(* IEC 61131-3 sources: plc-st-review/examples/state-machine, 14 files *)

(* ---- E_ConveyorState.st ---- *)
(*
 * Conveyor state machine enum.
 *
 * Used by FB_ConveyorState and (separately) by Conveyor_HMI. If we add a
 * value here and forget to handle it in the HMI's CASE, plc-st-review will
 * surface STATE_UNHANDLED.
 *)

TYPE E_ConveyorState :
    (IDLE := 0, STARTING, RUNNING, STOPPING, FAULT);
END_TYPE

(* ---- E_DiagMode.st ---- *)
(*
 * E_DiagMode — diagnostic verbosity levels for FB_AxisRamp.
 *
 * The demo PR removes DIAG_LEGACY (ENUM_VALUE_REMOVED) and drops the
 * DIAG_VERBOSE branch from FB_AxisRamp's CASE while keeping the value
 * in the enum (ENUM_VALUE_UNUSED).
 *)

TYPE E_DiagMode :
    (DIAG_OFF := 0, DIAG_BASIC, DIAG_VERBOSE, DIAG_LEGACY);
END_TYPE

(* ---- Globals.st ---- *)
(*
 * Globals for the conveyor demo.
 *
 * Demonstrates VAR_GLOBAL CONSTANT (constants the engine watches) and a
 * non-constant global (typed reference for callers).
 *)

VAR_GLOBAL CONSTANT
    SAFETY_TIMEOUT      : TIME := T#2s;
    LIMIT_MAX_SPEED     : INT  := 100;
    LIMIT_MIN_SPEED     : INT  := 5;
    CONVEYOR_SLOTS      : INT  := 10;
END_VAR

VAR_GLOBAL
    gFlowSetpoint       : REAL := 0.0;
END_VAR

(* ---- I_Diagnostic.st ---- *)
(*
 * I_Diagnostic — diagnostic contract implemented by FB_DiagUnit.
 *
 * The demo PR adds a second method (SelfTest) to this interface without
 * adding it to the implementer, surfacing METHOD_ADDED_TO_INTERFACE.
 *)

INTERFACE I_Diagnostic
METHOD Reset : BOOL
END_METHOD
END_INTERFACE

(* ---- FB_AxisRamp.st ---- *)
{attribute 'qualified_only'}
(*
 * FB_AxisRamp — ramps an axis toward a setpoint and counts cycles.
 *
 * The demo PR exercises five diff-based checks against this file:
 *   PRAGMA_CHANGED         the {attribute} pragma is swapped
 *   INHERITANCE_CHANGED    EXTENDS FB_Base -> FB_BaseV2
 *   ARRAY_BOUNDS_CHANGED   aHistory grows from [0..9] to [0..19]
 *   COUNTER_VALUE_CHANGED  cCycles.PV 100 -> 500
 *   ENUM_VALUE_UNUSED      the DIAG_VERBOSE CASE branch is removed
 *)

FUNCTION_BLOCK FB_AxisRamp EXTENDS FB_Base
VAR_INPUT
    rSetpoint : REAL;
    eMode     : E_DiagMode;
    xCount    : BOOL;
END_VAR
VAR_OUTPUT
    rPosition : REAL;
END_VAR
VAR
    aHistory  : ARRAY [0..9] OF REAL;
    cCycles   : CTU;
    iIndex    : INT;
END_VAR

cCycles(CU := xCount, PV := 100);

CASE eMode OF
    E_DiagMode.DIAG_OFF:
        rPosition := rSetpoint;
    E_DiagMode.DIAG_BASIC:
        rPosition := rSetpoint * 0.5;
    E_DiagMode.DIAG_VERBOSE:
        rPosition := rSetpoint * 0.25;
    E_DiagMode.DIAG_LEGACY:
        rPosition := 0.0;
END_CASE;

aHistory[iIndex] := rSetpoint;
END_FUNCTION_BLOCK

(* ---- FB_Base.st ---- *)
(*
 * FB_Base / FB_BaseV2 — base classes for the diagnostics demo.
 *
 * FB_AxisRamp EXTENDS FB_Base here; the demo PR re-points it at
 * FB_BaseV2 to surface INHERITANCE_CHANGED. Both are deliberately
 * trivial — they exist only to be inherited from.
 *)

FUNCTION_BLOCK FB_Base
VAR
    xInitialized : BOOL;
END_VAR
xInitialized := TRUE;
END_FUNCTION_BLOCK

FUNCTION_BLOCK FB_BaseV2
VAR
    xInitialized : BOOL;
    iRevision    : INT;
END_VAR
xInitialized := TRUE;
iRevision := 2;
END_FUNCTION_BLOCK

(* ---- FB_ConveyorState.st ---- *)
(*
 * FB_ConveyorState — minimal conveyor state machine.
 *
 * Implements a Mealy-style state machine over E_ConveyorState, with a
 * startup-delay timer and a configurable target speed. Designed to exercise
 * several plc-st-review checks at once when the file is edited.
 *)

FUNCTION_BLOCK FB_ConveyorState
VAR_INPUT
    xEnable             : BOOL;
    rTargetSpeed        : REAL;
END_VAR
VAR_OUTPUT
    eState              : E_ConveyorState;
    xRunning            : BOOL;
    rActualSpeed        : REAL;
END_VAR
VAR
    T_StartupDelay      : TON;
    iRamp               : INT;
END_VAR

(* Startup delay — driven by a TON instance. *)
T_StartupDelay(IN := (eState = E_ConveyorState.STARTING), PT := T#2s);

CASE eState OF
    E_ConveyorState.IDLE:
        IF xEnable THEN
            eState := E_ConveyorState.STARTING;
        END_IF;

    E_ConveyorState.STARTING:
        IF T_StartupDelay.Q THEN
            eState := E_ConveyorState.RUNNING;
            rActualSpeed := 0.0;
        END_IF;

    E_ConveyorState.RUNNING:
        xRunning := TRUE;
        (* Linear ramp toward target speed using a FOR loop. *)
        FOR iRamp := 1 TO CONVEYOR_SLOTS BY 1 DO
            rActualSpeed := rActualSpeed + (rTargetSpeed - rActualSpeed) * 0.1;
        END_FOR;
        IF NOT xEnable THEN
            eState := E_ConveyorState.STOPPING;
        END_IF;

    E_ConveyorState.STOPPING:
        xRunning := FALSE;
        rActualSpeed := 0.0;
        eState := E_ConveyorState.IDLE;

    E_ConveyorState.FAULT:
        xRunning := FALSE;
        rActualSpeed := 0.0;
END_CASE;

END_FUNCTION_BLOCK

(* ---- FB_DiagUnit.st ---- *)
(*
 * FB_DiagUnit — implements I_Diagnostic.
 *
 * The demo PR adds a SelfTest method to I_Diagnostic; this FB does NOT
 * gain a matching method, surfacing METHOD_ADDED_TO_INTERFACE.
 *)

FUNCTION_BLOCK FB_DiagUnit IMPLEMENTS I_Diagnostic
VAR
    xReady : BOOL;
END_VAR

METHOD Reset : BOOL
    xReady := FALSE;
    Reset := TRUE;
END_METHOD

xReady := TRUE;
END_FUNCTION_BLOCK

(* ---- FB_Legacy.st ---- *)
(*
 * FB_Legacy — a deprecated helper kept only so the demo PR can delete
 * the whole file and surface POU_DELETED. Nothing calls it.
 *)

FUNCTION_BLOCK FB_Legacy
VAR_INPUT
    xTrigger : BOOL;
END_VAR
VAR_OUTPUT
    xDone : BOOL;
END_VAR
xDone := xTrigger;
END_FUNCTION_BLOCK

(* ---- FB_LineController.st ---- *)
(*
 * FB_LineController - top-level conveyor-line coordinator.
 *
 * A deliberately involved orchestrator: it sequences the axis ramp, the speed
 * estimate, the diagnostic unit and the metrics helper behind layered mode and
 * guard logic. It exists so the --metrics report has a realistic
 * high-complexity hub to rank (it lands in the red band), and so the blocks it
 * drives are reported as live rather than dead code. The body is intentionally
 * tangled but otherwise clean - it triggers no review findings on its own.
 *)

FUNCTION_BLOCK FB_LineController EXTENDS FB_BaseV2
VAR_INPUT
    xRun        : BOOL;
    iMode       : INT;
    rSetpoint   : REAL;
    iPulses     : INT;
    xManual     : BOOL;
END_VAR
VAR_OUTPUT
    rLineSpeed  : REAL;
    xActive     : BOOL;
    iFaultCode  : INT;
END_VAR
VAR
    fbRamp      : FB_AxisRamp;
    fbSpeed     : FB_SpeedCalc;
    fbDiag      : FB_DiagUnit;
    fbMetrics   : FB_MetricsDemo;
    T_Settle    : TON;
    rLocalSpeed : REAL;
    iStep       : INT;
    iGuard      : INT;
    iFault      : INT;
END_VAR

(* Sub-blocks run every scan; their outputs feed the mode logic below. *)
fbSpeed(iPulseCount := iPulses, rScale := 0.5);
fbDiag();
T_Settle(IN := xRun, PT := T#500ms);

CASE iMode OF
    0:  (* idle - wait for a run request that isn't a manual hold *)
        IF xRun AND NOT xManual THEN
            iStep := 1;
        ELSIF xManual THEN
            iStep := 0;
        END_IF;

    1:  (* ramping - climb toward setpoint once the settle timer elapses *)
        IF T_Settle.Q THEN
            fbRamp(rSetpoint := rSetpoint, eMode := E_DiagMode.DIAG_BASIC, xCount := xRun);
            FOR iGuard := 1 TO CONVEYOR_SLOTS BY 1 DO
                IF fbSpeed.rSpeed > rLocalSpeed THEN
                    rLocalSpeed := rLocalSpeed + (rSetpoint - rLocalSpeed) * 0.1;
                    IF rLocalSpeed > LIMIT_MAX_SPEED THEN
                        rLocalSpeed := LIMIT_MAX_SPEED;
                    END_IF;
                    IF xManual OR iGuard > LIMIT_MIN_SPEED THEN
                        iStep := iGuard;
                    END_IF;
                END_IF;
            END_FOR;
        END_IF;

    2:  (* running - advance the line, sampling metrics as it goes *)
        WHILE iStep < CONVEYOR_SLOTS AND xRun DO
            iStep := iStep + 1;
            IF rLocalSpeed >= rSetpoint THEN
                EXIT;
            END_IF;
            IF iStep >= LIMIT_MIN_SPEED THEN
                fbMetrics(x := iStep);
                IF fbMetrics.y > 0 OR xManual THEN
                    rLocalSpeed := fbRamp.rPosition;
                END_IF;
            END_IF;
        END_WHILE;

    3:  (* diagnostics - classify the speed estimate into a fault code *)
        IF fbSpeed.rSpeed < LIMIT_MIN_SPEED THEN
            iFault := 1;
        ELSIF fbSpeed.rSpeed > LIMIT_MAX_SPEED THEN
            iFault := 2;
        ELSE
            iFault := 0;
        END_IF;

    4:  (* hold - manual override parks the line *)
        IF xManual THEN
            iStep := 0;
            rLocalSpeed := 0.0;
        END_IF;

    ELSE
        iStep := 0;
END_CASE;

IF iFault > 0 THEN
    xActive := FALSE;
ELSIF xRun THEN
    xActive := TRUE;
END_IF;

rLineSpeed := rLocalSpeed;
iFaultCode := iFault;
END_FUNCTION_BLOCK

(* ---- FB_MetricsDemo.st ---- *)
// Baseline version of the metrics-demo block. The demo PR (#1) ships a
// heavily expanded version of this same FB, so the diff exercises the
// metric-regression checks (COMPLEXITY_INCREASED, NESTING_INCREASED,
// LOC_SPIKE) without disturbing any other fixture.
FUNCTION_BLOCK FB_MetricsDemo
VAR_INPUT
    x : INT;
END_VAR
VAR_OUTPUT
    y : INT;
END_VAR
y := x;
END_FUNCTION_BLOCK

(* ---- FB_SpeedCalc.st ---- *)
(*
 * FB_SpeedCalc — converts a raw pulse count to a speed estimate.
 *
 * The demo PR renames this POU to FB_SpeedCalculator (keeping the exact
 * same input/output signature) to surface POU_RENAMED.
 *)

FUNCTION_BLOCK FB_SpeedCalc
VAR_INPUT
    iPulseCount : INT;
    rScale      : REAL;
END_VAR
VAR_OUTPUT
    rSpeed      : REAL;
END_VAR
VAR
    rRaw        : REAL;
END_VAR
rRaw := rScale;
IF iPulseCount > 0 THEN
    rSpeed := rRaw;
ELSE
    rSpeed := 0.0;
END_IF;
END_FUNCTION_BLOCK

(* ---- FB_Watchdog.st ---- *)
(*
 * FB_Watchdog — trivial heartbeat monitor.
 *
 * The demo PR changes ONLY the inline comment below, leaving the AST
 * structurally identical between revisions, to surface COMMENT_ONLY.
 *)

FUNCTION_BLOCK FB_Watchdog
VAR_INPUT
    xHeartbeat : BOOL;
END_VAR
VAR_OUTPUT
    xAlive : BOOL;
END_VAR
(* heartbeat is forwarded straight through *)
xAlive := xHeartbeat;
END_FUNCTION_BLOCK

(* ---- Conveyor_HMI.st ---- *)
(*
 * Conveyor_HMI — display formatter for the conveyor state machine.
 *
 * Lives in a different file than FB_ConveyorState on purpose: the engine's
 * cross-file analysis is what surfaces STATE_UNHANDLED when the enum gains
 * a value and only one of the CASE statements is updated.
 *)

PROGRAM Conveyor_HMI
VAR
    fbConveyor          : FB_ConveyorState;
    fbLine              : FB_LineController;
    sStateLabel         : STRING := '';
END_VAR

fbConveyor(xEnable := TRUE, rTargetSpeed := 50.0);
fbLine(xRun := TRUE, iMode := 1, rSetpoint := 50.0, iPulses := 100, xManual := FALSE);

CASE fbConveyor.eState OF
    E_ConveyorState.IDLE:       sStateLabel := 'Idle';
    E_ConveyorState.STARTING:   sStateLabel := 'Starting...';
    E_ConveyorState.RUNNING:    sStateLabel := 'Running';
    E_ConveyorState.STOPPING:   sStateLabel := 'Stopping...';
    E_ConveyorState.FAULT:      sStateLabel := 'FAULT';
END_CASE;

END_PROGRAM
